ABB RAPID module: traj5.MOD

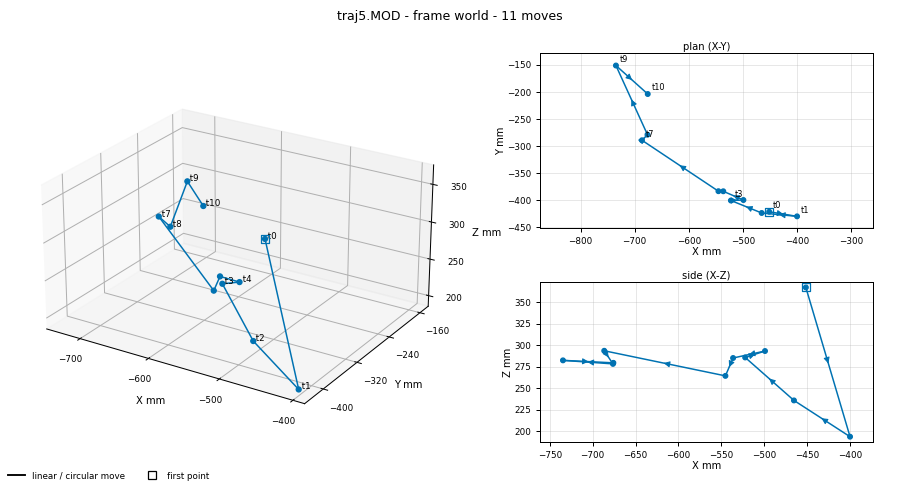
[picture p0: tool path of traj5.MOD in frame world, 11 of 12 moves have a stored position in this frame; points joined in program order, loops and branches not executed]
MODULE MainModule
PERS tooldata Servo:=[TRUE,[[0,0,114.2],[1,0,0,0]],[0.215,[8.7,12.3,49.2],[1,0,0,0],0.00021,0.00024,0.00009]];
PERS tooldata tObject:=[TRUE,[[0,0,130],[0.707106781,-0.707106781,0,0]],[0.215,[8.7,12.3,49.2],[1,0,0,0],0.00021,0.00024,0.00009]];


PERS wobjdata handpos:= [FALSE,TRUE,"",[[-400,0,250],[ 0.319436873,  0.370938549, -0.871988920, 0.0]],[[0,0,0],[1,0,0,0]]];
    PROC main()
        ConfL\Off;
        SingArea\Wrist;
        !Startpos
        MoveAbsJ [[0.441359,-16.418,10.8814,2.79121,60.2034,-14.3875],[168.362,9E+09,9E+09,9E+09,9E+09,9E+09]] \NoEOffs, v1000, fine, wi_tGripper;
        path;
    ENDPROC
    PROC path()

VAR robtarget t0 := [[364.6408440533277, -243.92922019584628, 35.06858647183071], [0,1,0,0], [0,0,-1,4], [-96,9E+09,9E+09,9E+09,9E+09,9E+09]];
VAR robtarget t1 := [[246.44845023422806, -324.58408470244, 146.7954967805132], [0,1,0,0], [0,0,-1,4], [-96,9E+09,9E+09,9E+09,9E+09,9E+09]];
VAR robtarget t2 := [[299.9812714790488, -267.7868316047999, 148.08487039368015], [0,1,0,0], [0,0,-1,4], [-96,9E+09,9E+09,9E+09,9E+09,9E+09]];
VAR robtarget t3 := [[342.55596986528303, -202.48710137708892, 134.4356752151807], [0,1,0,0], [0,0,-1,4], [-96,9E+09,9E+09,9E+09,9E+09,9E+09]];
VAR robtarget t4 := [[334.1175393307455, -214.9854154213677, 115.3982124665365], [0,1,0,0], [0,0,-1,4], [-96,9E+09,9E+09,9E+09,9E+09,9E+09]];
VAR robtarget t5 := [[338.51303085539655, -181.15294473070082, 138.76147952204838], [0,1,0,0], [0,0,-1,4], [-96,9E+09,9E+09,9E+09,9E+09,9E+09]];
VAR robtarget t6 := [[331.4922083584789, -180.2109910647929, 160.26885062581596], [0,1,0,0], [0,0,-1,4], [-96,9E+09,9E+09,9E+09,9E+09,9E+09]];
VAR robtarget t7 := [[360.44006530927606, -13.776016261393188, 193.3519395014274], [0,1,0,0], [0,0,-1,4], [-96,9E+09,9E+09,9E+09,9E+09,9E+09]];
VAR robtarget t8 := [[339.98570309289084, -16.524397167637353, 197.42248809944851], [0,1,0,0], [0,0,-1,4], [-96,9E+09,9E+09,9E+09,9E+09,9E+09]];
VAR robtarget t9 := [[289.9854386293305, 114.70228205129987, 196.3186015345908], [0,1,0,0], [0,0,-1,4], [-96,9E+09,9E+09,9E+09,9E+09,9E+09]];
VAR robtarget t10 := [[291.8208398529501, 37.89718547825187, 178.3605999717464], [0,1,0,0], [0,0,-1,4], [-96,9E+09,9E+09,9E+09,9E+09,9E+09]];

MoveL t0, v100\V:=100.000, z1, wi_tGripper, \WObj:=handpos;
MoveL t1, v100\V:=100.000, z1, wi_tGripper, \WObj:=handpos;
MoveL t2, v100\V:=100.000, z1, wi_tGripper, \WObj:=handpos;
MoveL t3, v100\V:=100.000, z1, wi_tGripper, \WObj:=handpos;
MoveL t4, v100\V:=100.000, z1, wi_tGripper, \WObj:=handpos;
MoveL t5, v100\V:=100.000, z1, wi_tGripper, \WObj:=handpos;
MoveL t6, v100\V:=100.000, z1, wi_tGripper, \WObj:=handpos;
MoveL t7, v100\V:=100.000, z1, wi_tGripper, \WObj:=handpos;
MoveL t8, v100\V:=100.000, z1, wi_tGripper, \WObj:=handpos;
MoveL t9, v100\V:=100.000, z1, wi_tGripper, \WObj:=handpos;
MoveL t10, v100\V:=100.000, z1, wi_tGripper, \WObj:=handpos;



ENDPROC
ENDMODULE
